{attribute addProperty BoxType "EP5001-0002-0016"}
{attribute addProperty Id "SSI_InputsAT %I*SSI_Inputs_C03DB35B4860WcStateAT %I*WcState_98A4DF7520.250InfoDataAT %I*InfoData_BC63D37F80100"}
{attribute addProperty CRC "1006069159"}
{attribute addProperty SizeInBites "130"}
{attribute addProperty SizeInBytes "16.25"}
TYPE EP5001_99FC62FA :
STRUCT
	{attribute addProperty Name "SSI_Inputs"}
	SSI_Inputs : SSI_Inputs_C03DB35B;
	{attribute addProperty Name "WcState"}
	WcState : WcState_98A4DF75;
	{attribute addProperty Name "InfoData"}
	InfoData : InfoData_BC63D37F;
END_STRUCT
END_TYPE

(* stored: Version 1.2.0.0, ProductVersion 3.1.4024.9
   DUT EP5001_99FC62FA: Id {2b4be844-5636-4a6e-8c85-ae068539f4b8} *)
